// TwinCAT 3 PLC project Lamppu1
// ProgramVersion: 3.1.4026.10
// CompilerDefines: VISU_USEPROPERTYINFO
// libraries:
//   Tc2_Standard, * (Beckhoff Automation GmbH)
//   Tc2_System, * (Beckhoff Automation GmbH)
//   VisuSymbols, 4.5.0.0 (System)
// project tree:
//   / GlobalTextList.TcGTLO, PlcTask.TcTTO, Visualization Manager.TcVMO (not stored)
//   POUs/ MAIN.TcPOU
//   VISUs/ Visualization.TcVIS
// real-time tasks:
//   TASK PlcTask: cycle T#10ms, priority 20, ADS port 350

CONFIGURATION Lamppu1
    RESOURCE PLC ON TwinCAT3
        TASK PlcTask(INTERVAL := T#10ms, PRIORITY := 20);
        PROGRAM MAIN WITH PlcTask : MAIN;
    END_RESOURCE
END_CONFIGURATION

// ---- POUs/MAIN.TcPOU
PROGRAM MAIN
VAR
	_LampIsOn		: BOOL := FALSE;
	_ButtonIsPushed	: BOOL := FALSE;
END_VAR

// This program operates a lamp. When a button is pushed, and held down, the lamp turns on.
// When the button is released, the lamp turns off. Instead of using a real lamp and a button,
// they are in the visualization.

IF _ButtonIsPushed THEN
	_LampIsOn := TRUE;
ELSE
	_LampIsOn := FALSE;
END_IF

END_PROGRAM

// ---- GlobalTextList.TcGTLO
TEXTLIST GlobalTextList
  938 = 'Push to light the lamp'
  231 = 'This here is a button'
END_TEXTLIST

// ---- VISUs/Visualization.TcVIS
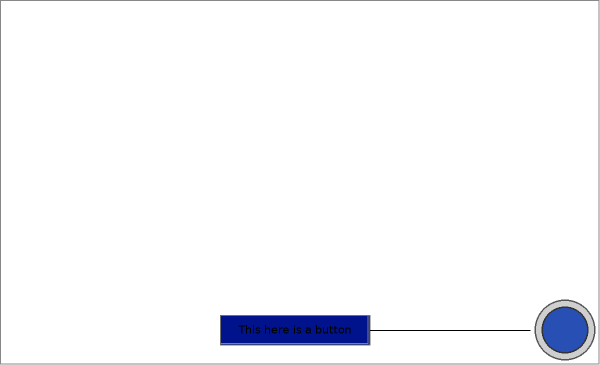
VISUALIZATION Visualization  // 600x365
    Button (220,315 150x30), "This here is a button", tooltip "Push to light the lamp"
        OnMouseDown: toggle MAIN._ButtonIsPushed
        OnMouseUp: toggle MAIN._ButtonIsPushed
    Lamp1 (530,295 70x70), variable: MAIN._LampIsOn, style: Lamp-Lamp1-Blue
    Line (370,330) (530,330)
END_VISUALIZATION
